(* Logix 5000 project; controller BTS01 vendor 1 type 14 code 217 rev 32.14; software revision 32.04; part 3 of 15 *)
(* tags used below, declared in another part *)
   AG1101 : DTE_VFD;   // Tank 1100 Agitator
   AG1201 : DTE_VFD;   // Tank 1200 Agitator
   Alarm_Active : DINT;
   Alarm_TMR : TIMER[17,32];
   ALM_ENABLE : DINT[25];
   C02S01 : REAL[8];   // 5069-IF8
   C02S03 : INT;   // 5069-IB16
   C02S06 : INT;   // 5069-IB16
   CIP_1_ACTIVE_CIRCUIT : DINT;
   CIP_1_Circuit1_Prox_Mismatch : BOOL;
   CIP_1_Circuit1_Tank_Not_Empty : BOOL;
   CIP_1_Circuit2_Prox_Mismatch : BOOL;
   CIP_1_Circuit2_Tank_Not_Empty : BOOL;
   CIP_1_Circuit3_Prox_Mismatch : BOOL;
   CIP_1_Circuit4_Prox_Mismatch : BOOL;
   CIP_1_SEQ_CTU : COUNTER;   // CIP 1 SEQUENCE STEP COUNTER THIS IS THE SEQUENCE STEP CONTROL
   CIP_1_START_PB_HMI : BOOL;
   CIP_Cart_Comm_Failed : BOOL;
   HMI_Global_Alarm_Ack_PB : BOOL;
   HMIAlarms : DINT[25];   // Alarm Trigger Array
   HMIAlarmsMsg : STRING64[17,32];   // Alarm Descriptions to Match Alarm Trigger Array
   P1001 : DTE_VFD;   // Dressing Tank Fill Pump
   P1002 : DTE_VFD;   // Product Filler Fill Pump
   P1003 : DTE_VFD;   // CIP Return Pump
   P1004 : DTE_VFD;   // Filler CIP Return Pump

   V1007_CIP_ENABLE : BOOL;
   V1007_CIP_PULSE : BOOL;
   V1007_Desc : STRING;
   V1007_PIDName : STRING;
   V1101 : DTE_Air_Valve_v2 := (CMD := 1, OUT := 1, ALM_PRE := 7000, P := 1, M := 2, Allowed := 1, Status := 1, ITEMTAG := 1101, MOA_Mode := 1);   // Tank 1100 Fill Valve
   V1101_CIP_ENABLE : BOOL;
   V1101_CIP_PULSE : BOOL;
   V1101_Desc : STRING;
   V1101_PIDName : STRING;
   V1102 : DTE_Air_Valve_v2 := (ALM_PRE := 7000, M := 2, Allowed := 1, ITEMTAG := 1102, MOA_Mode := 1);   // Tank 1100 Discharge Valve
   V1102_CIP_ENABLE : BOOL;
   V1102_CIP_PULSE : BOOL;
   V1102_Desc : STRING;
   V1102_PIDName : STRING;
   V1103 : DTE_Air_Valve_v2 := (ALM_PRE := 7000, M := 2, Allowed := 1, ITEMTAG := 1103, MOA_Mode := 1);   // Tank 1100 Line Valve
   V1103_CIP_ENABLE : BOOL;
   V1103_CIP_PULSE : BOOL;
   V1103_Desc : STRING;
   V1103_PIDName : STRING;
   V1201 : DTE_Air_Valve_v2 := (TOFF_OUT_ACC := 1, ALM_PRE := 7000, M := 2, Allowed := 1, ITEMTAG := 1201, MOA_Mode := 1);   // Tank 1200 Fill Valve
   V1201_CIP_ENABLE : BOOL;
   V1201_CIP_PULSE : BOOL;
   V1201_Desc : STRING;
   V1201_PIDName : STRING;
   V1202 : DTE_Air_Valve_v2 := (ALM_PRE := 7000, M := 2, Allowed := 1, ITEMTAG := 1202, MOA_Mode := 1);   // Tank 1200 Discharge Valve
   V1202_CIP_ENABLE : BOOL;
   V1202_CIP_PULSE : BOOL;
   V1202_Desc : STRING;
   V1202_PIDName : STRING;
   V1203 : DTE_Air_Valve_v2 := (ALM_PRE := 7000, M := 2, Allowed := 1, ITEMTAG := 1203, MOA_Mode := 1);   // Tank 1200 Line Valve
   V1203_CIP_ENABLE : BOOL;
   V1203_CIP_PULSE : BOOL;
   V1203_Desc : STRING;
   V1203_PIDName : STRING;
   VFD1001_SCP : DTE_SCP_W_LIM := (Input_Max := 100.0, Scaled_Max := 100.0, Limit_En := 1);   // Bowl Chopper Disc Speed Reference
   VFD1002_SCP : DTE_SCP_W_LIM := (Input_Max := 100.0, Scaled_Max := 100.0, Limit_En := 1);   // Dressing Tank Disc Speed Reference
   VFD1003_SCP : DTE_SCP_W_LIM := (Input_Max := 100.0, Scaled_Max := 100.0, Limit_En := 1);   // CIP Return Pump Speed Reference
   VFD1004_SCP : DTE_SCP_W_LIM := (Input_Max := 100.0, Scaled_Max := 100.0, Limit_En := 1);   // Filler CIP Return Pump Speed Reference
   VFD1101_SCP : DTE_SCP_W_LIM := (Input_Max := 100.0, Scaled_Max := 100.0, Limit_En := 1);   // Tank 1100 Agitator Speed Reference
   VFD1201_SCP : DTE_SCP_W_LIM := (Input_Max := 100.0, Scaled_Max := 100.0, Limit_En := 1);   // Tank 1200 Agitator Speed Reference
   ZS1000_1_Ind : DINT;
   ZS1000_2_Ind : DINT;
   ZS1000_3_Ind : DINT;
   ZS1000_4_Ind : DINT := 3;
   ZS1000_5_Ind : DINT;
   ZS1001_1_Ind : DINT;
   ZS1001_2_Ind : DINT;
   ZS1001_3_Ind : DINT;
   ZS1001_4_Ind : DINT;
   ZS1001_5_Ind : DINT := 3;
   ZS1101_Ind : DINT;
   ZS1201_Ind : DINT;
END_VAR

PROGRAM Alarm   (* main routine Alarm_Main *)

ROUTINE Alarm_00   (* ladder *)
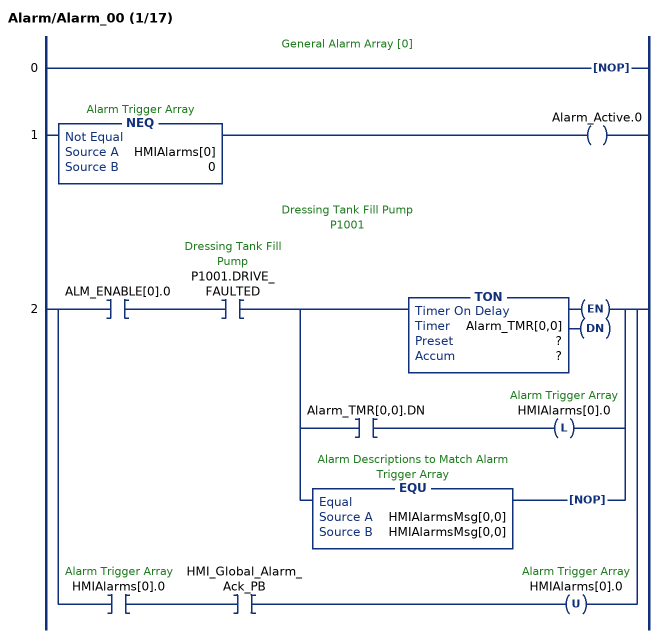
   // General Alarm Array [0]
   0: NOP();
   1: NEQ(HMIAlarms[0],0)OTE(Alarm_Active.0);
   // Dressing Tank Fill Pump
   // P1001
   2: [XIC(ALM_ENABLE[0].0) XIC(P1001.DRIVE_FAULTED) [TON(Alarm_TMR[0,0],?,?) ,XIC(Alarm_TMR[0,0].DN) OTL(HMIAlarms[0].0) ,EQU(HMIAlarmsMsg[0,0],HMIAlarmsMsg[0,0]) NOP() ] ,XIC(HMIAlarms[0].0) XIC(HMI_Global_Alarm_Ack_PB) OTU(HMIAlarms[0].0) ];
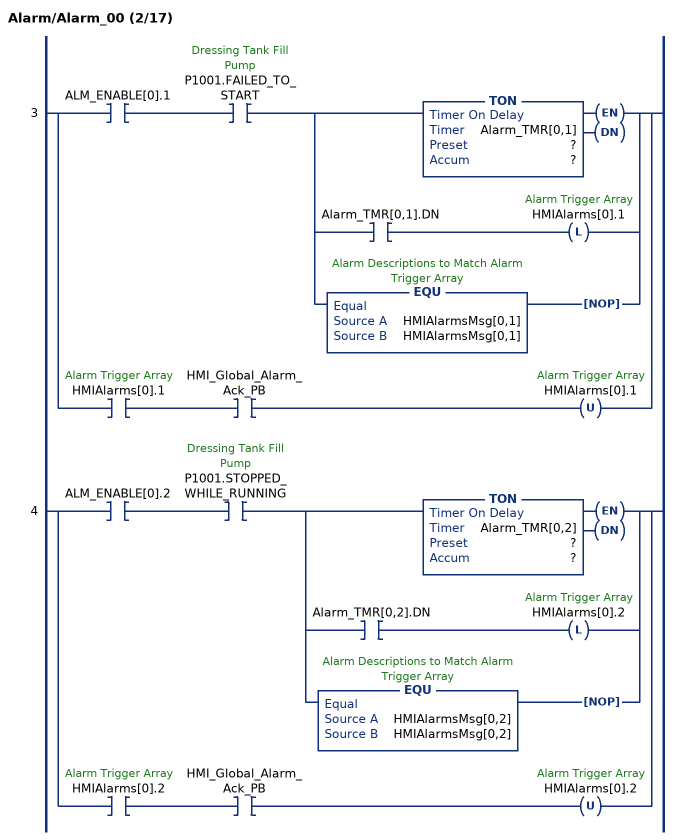
   3: [XIC(ALM_ENABLE[0].1) XIC(P1001.FAILED_TO_START) [TON(Alarm_TMR[0,1],?,?) ,XIC(Alarm_TMR[0,1].DN) OTL(HMIAlarms[0].1) ,EQU(HMIAlarmsMsg[0,1],HMIAlarmsMsg[0,1]) NOP() ] ,XIC(HMIAlarms[0].1) XIC(HMI_Global_Alarm_Ack_PB) OTU(HMIAlarms[0].1) ];
   4: [XIC(ALM_ENABLE[0].2) XIC(P1001.STOPPED_WHILE_RUNNING) [TON(Alarm_TMR[0,2],?,?) ,XIC(Alarm_TMR[0,2].DN) OTL(HMIAlarms[0].2) ,EQU(HMIAlarmsMsg[0,2],HMIAlarmsMsg[0,2]) NOP() ] ,XIC(HMIAlarms[0].2) XIC(HMI_Global_Alarm_Ack_PB) OTU(HMIAlarms[0].2) ];
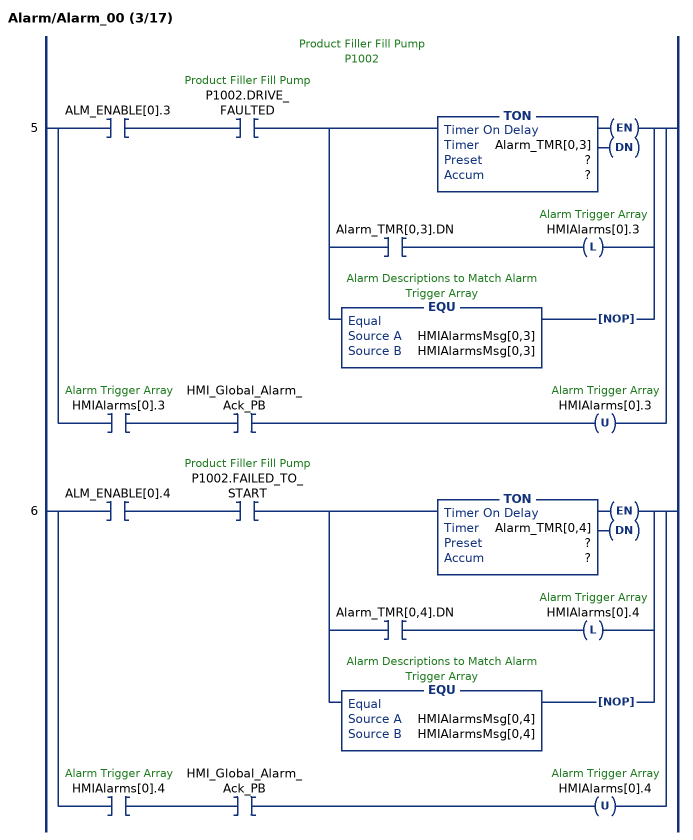
   // Product Filler Fill Pump
   // P1002
   5: [XIC(ALM_ENABLE[0].3) XIC(P1002.DRIVE_FAULTED) [TON(Alarm_TMR[0,3],?,?) ,XIC(Alarm_TMR[0,3].DN) OTL(HMIAlarms[0].3) ,EQU(HMIAlarmsMsg[0,3],HMIAlarmsMsg[0,3]) NOP() ] ,XIC(HMIAlarms[0].3) XIC(HMI_Global_Alarm_Ack_PB) OTU(HMIAlarms[0].3) ];
   6: [XIC(ALM_ENABLE[0].4) XIC(P1002.FAILED_TO_START) [TON(Alarm_TMR[0,4],?,?) ,XIC(Alarm_TMR[0,4].DN) OTL(HMIAlarms[0].4) ,EQU(HMIAlarmsMsg[0,4],HMIAlarmsMsg[0,4]) NOP() ] ,XIC(HMIAlarms[0].4) XIC(HMI_Global_Alarm_Ack_PB) OTU(HMIAlarms[0].4) ];
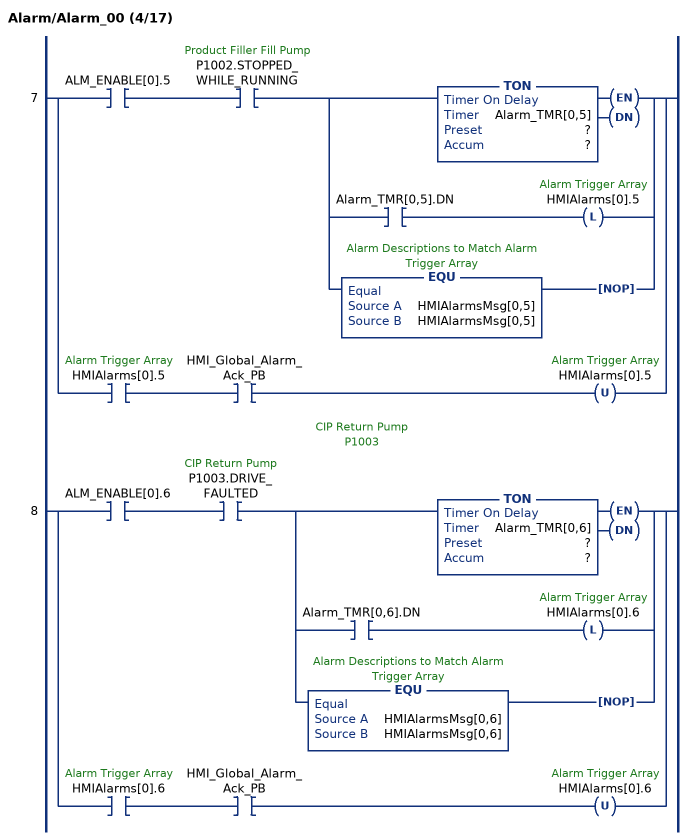
   7: [XIC(ALM_ENABLE[0].5) XIC(P1002.STOPPED_WHILE_RUNNING) [TON(Alarm_TMR[0,5],?,?) ,XIC(Alarm_TMR[0,5].DN) OTL(HMIAlarms[0].5) ,EQU(HMIAlarmsMsg[0,5],HMIAlarmsMsg[0,5]) NOP() ] ,XIC(HMIAlarms[0].5) XIC(HMI_Global_Alarm_Ack_PB) OTU(HMIAlarms[0].5) ];
   // CIP Return Pump
   // P1003
   8: [XIC(ALM_ENABLE[0].6) XIC(P1003.DRIVE_FAULTED) [TON(Alarm_TMR[0,6],?,?) ,XIC(Alarm_TMR[0,6].DN) OTL(HMIAlarms[0].6) ,EQU(HMIAlarmsMsg[0,6],HMIAlarmsMsg[0,6]) NOP() ] ,XIC(HMIAlarms[0].6) XIC(HMI_Global_Alarm_Ack_PB) OTU(HMIAlarms[0].6) ];
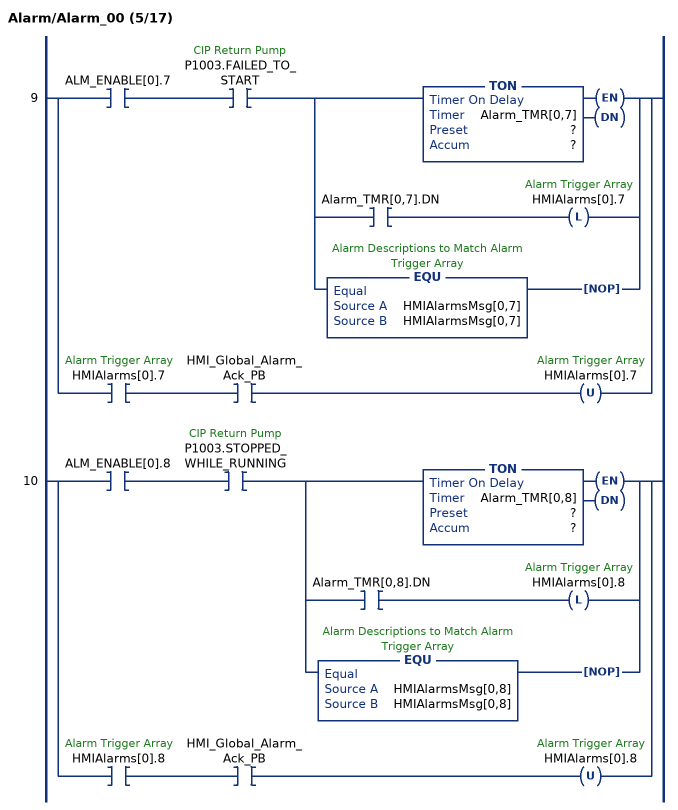
   9: [XIC(ALM_ENABLE[0].7) XIC(P1003.FAILED_TO_START) [TON(Alarm_TMR[0,7],?,?) ,XIC(Alarm_TMR[0,7].DN) OTL(HMIAlarms[0].7) ,EQU(HMIAlarmsMsg[0,7],HMIAlarmsMsg[0,7]) NOP() ] ,XIC(HMIAlarms[0].7) XIC(HMI_Global_Alarm_Ack_PB) OTU(HMIAlarms[0].7) ];
   10: [XIC(ALM_ENABLE[0].8) XIC(P1003.STOPPED_WHILE_RUNNING) [TON(Alarm_TMR[0,8],?,?) ,XIC(Alarm_TMR[0,8].DN) OTL(HMIAlarms[0].8) ,EQU(HMIAlarmsMsg[0,8],HMIAlarmsMsg[0,8]) NOP() ] ,XIC(HMIAlarms[0].8) XIC(HMI_Global_Alarm_Ack_PB) OTU(HMIAlarms[0].8) ];
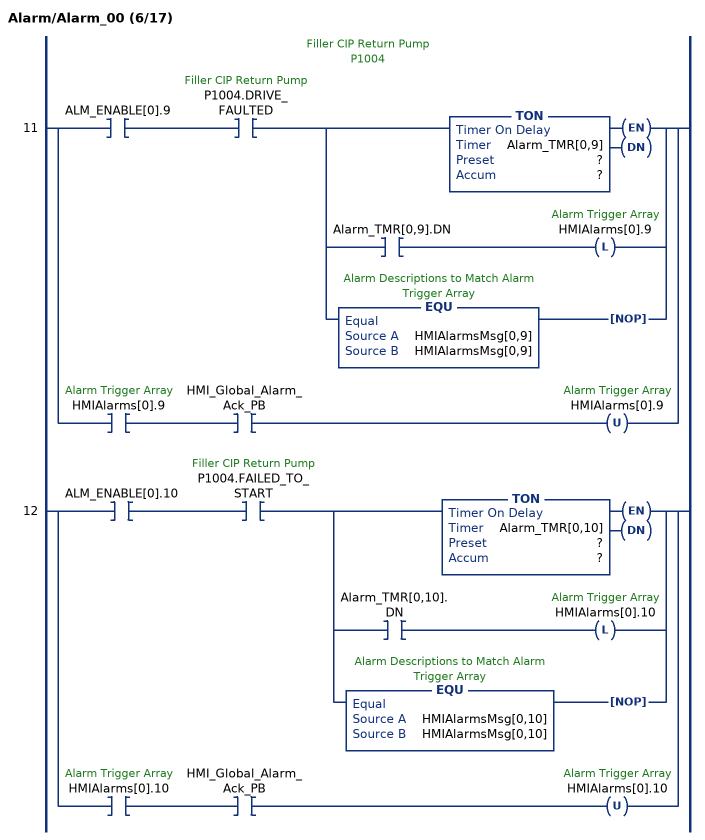
   // Filler CIP Return Pump
   // P1004
   11: [XIC(ALM_ENABLE[0].9) XIC(P1004.DRIVE_FAULTED) [TON(Alarm_TMR[0,9],?,?) ,XIC(Alarm_TMR[0,9].DN) OTL(HMIAlarms[0].9) ,EQU(HMIAlarmsMsg[0,9],HMIAlarmsMsg[0,9]) NOP() ] ,XIC(HMIAlarms[0].9) XIC(HMI_Global_Alarm_Ack_PB) OTU(HMIAlarms[0].9) ];
   12: [XIC(ALM_ENABLE[0].10) XIC(P1004.FAILED_TO_START) [TON(Alarm_TMR[0,10],?,?) ,XIC(Alarm_TMR[0,10].DN) OTL(HMIAlarms[0].10) ,EQU(HMIAlarmsMsg[0,10],HMIAlarmsMsg[0,10]) NOP() ] ,XIC(HMIAlarms[0].10) XIC(HMI_Global_Alarm_Ack_PB) OTU(HMIAlarms[0].10) ];
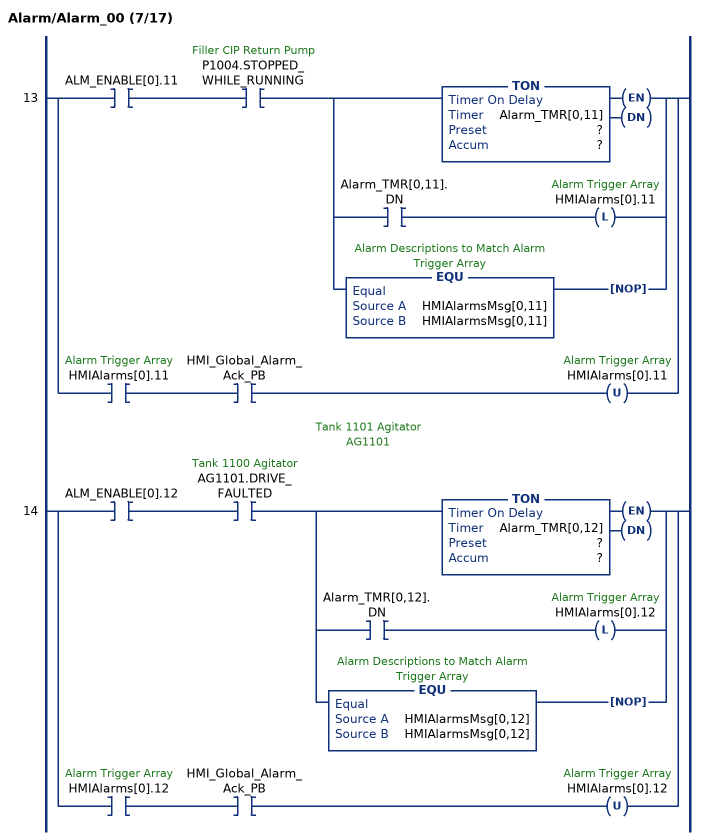
   13: [XIC(ALM_ENABLE[0].11) XIC(P1004.STOPPED_WHILE_RUNNING) [TON(Alarm_TMR[0,11],?,?) ,XIC(Alarm_TMR[0,11].DN) OTL(HMIAlarms[0].11) ,EQU(HMIAlarmsMsg[0,11],HMIAlarmsMsg[0,11]) NOP() ] ,XIC(HMIAlarms[0].11) XIC(HMI_Global_Alarm_Ack_PB) OTU(HMIAlarms[0].11) ];
   // Tank 1101 Agitator
   // AG1101
   14: [XIC(ALM_ENABLE[0].12) XIC(AG1101.DRIVE_FAULTED) [TON(Alarm_TMR[0,12],?,?) ,XIC(Alarm_TMR[0,12].DN) OTL(HMIAlarms[0].12) ,EQU(HMIAlarmsMsg[0,12],HMIAlarmsMsg[0,12]) NOP() ] ,XIC(HMIAlarms[0].12) XIC(HMI_Global_Alarm_Ack_PB) OTU(HMIAlarms[0].12) ];
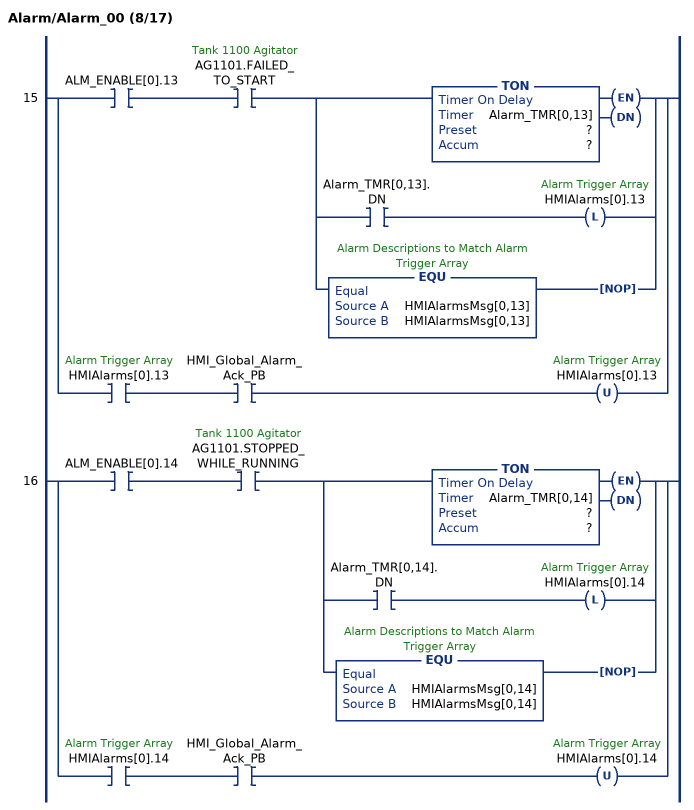
   15: [XIC(ALM_ENABLE[0].13) XIC(AG1101.FAILED_TO_START) [TON(Alarm_TMR[0,13],?,?) ,XIC(Alarm_TMR[0,13].DN) OTL(HMIAlarms[0].13) ,EQU(HMIAlarmsMsg[0,13],HMIAlarmsMsg[0,13]) NOP() ] ,XIC(HMIAlarms[0].13) XIC(HMI_Global_Alarm_Ack_PB) OTU(HMIAlarms[0].13) ];
   16: [XIC(ALM_ENABLE[0].14) XIC(AG1101.STOPPED_WHILE_RUNNING) [TON(Alarm_TMR[0,14],?,?) ,XIC(Alarm_TMR[0,14].DN) OTL(HMIAlarms[0].14) ,EQU(HMIAlarmsMsg[0,14],HMIAlarmsMsg[0,14]) NOP() ] ,XIC(HMIAlarms[0].14) XIC(HMI_Global_Alarm_Ack_PB) OTU(HMIAlarms[0].14) ];
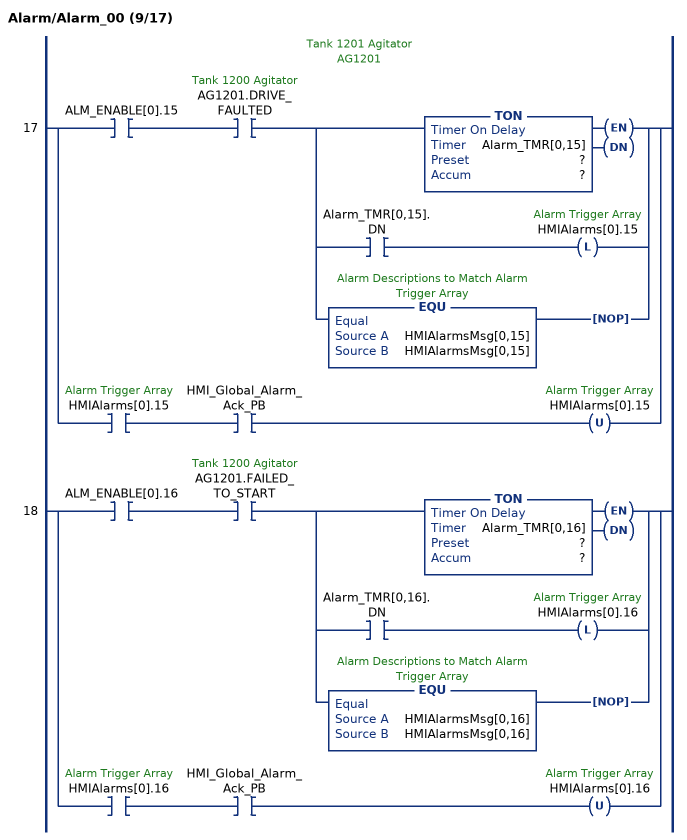
   // Tank 1201 Agitator
   // AG1201
   17: [XIC(ALM_ENABLE[0].15) XIC(AG1201.DRIVE_FAULTED) [TON(Alarm_TMR[0,15],?,?) ,XIC(Alarm_TMR[0,15].DN) OTL(HMIAlarms[0].15) ,EQU(HMIAlarmsMsg[0,15],HMIAlarmsMsg[0,15]) NOP() ] ,XIC(HMIAlarms[0].15) XIC(HMI_Global_Alarm_Ack_PB) OTU(HMIAlarms[0].15) ];
   18: [XIC(ALM_ENABLE[0].16) XIC(AG1201.FAILED_TO_START) [TON(Alarm_TMR[0,16],?,?) ,XIC(Alarm_TMR[0,16].DN) OTL(HMIAlarms[0].16) ,EQU(HMIAlarmsMsg[0,16],HMIAlarmsMsg[0,16]) NOP() ] ,XIC(HMIAlarms[0].16) XIC(HMI_Global_Alarm_Ack_PB) OTU(HMIAlarms[0].16) ];
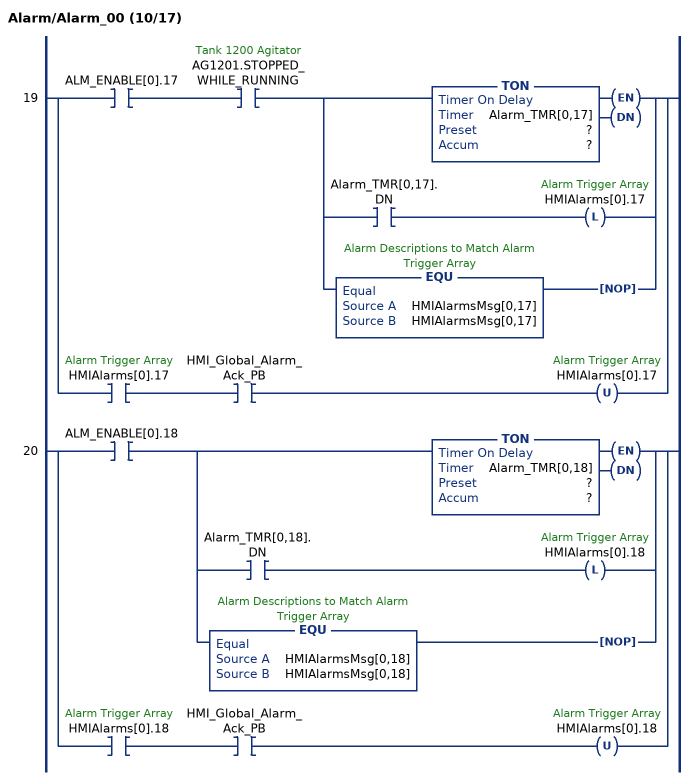
   19: [XIC(ALM_ENABLE[0].17) XIC(AG1201.STOPPED_WHILE_RUNNING) [TON(Alarm_TMR[0,17],?,?) ,XIC(Alarm_TMR[0,17].DN) OTL(HMIAlarms[0].17) ,EQU(HMIAlarmsMsg[0,17],HMIAlarmsMsg[0,17]) NOP() ] ,XIC(HMIAlarms[0].17) XIC(HMI_Global_Alarm_Ack_PB) OTU(HMIAlarms[0].17) ];
   20: [XIC(ALM_ENABLE[0].18) [TON(Alarm_TMR[0,18],?,?) ,XIC(Alarm_TMR[0,18].DN) OTL(HMIAlarms[0].18) ,EQU(HMIAlarmsMsg[0,18],HMIAlarmsMsg[0,18]) NOP() ] ,XIC(HMIAlarms[0].18) XIC(HMI_Global_Alarm_Ack_PB) OTU(HMIAlarms[0].18) ];
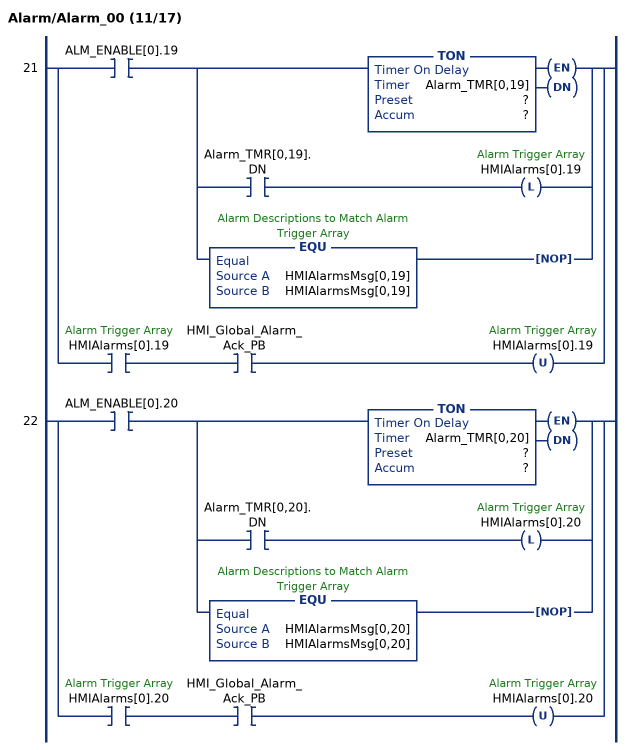
   21: [XIC(ALM_ENABLE[0].19) [TON(Alarm_TMR[0,19],?,?) ,XIC(Alarm_TMR[0,19].DN) OTL(HMIAlarms[0].19) ,EQU(HMIAlarmsMsg[0,19],HMIAlarmsMsg[0,19]) NOP() ] ,XIC(HMIAlarms[0].19) XIC(HMI_Global_Alarm_Ack_PB) OTU(HMIAlarms[0].19) ];
   22: [XIC(ALM_ENABLE[0].20) [TON(Alarm_TMR[0,20],?,?) ,XIC(Alarm_TMR[0,20].DN) OTL(HMIAlarms[0].20) ,EQU(HMIAlarmsMsg[0,20],HMIAlarmsMsg[0,20]) NOP() ] ,XIC(HMIAlarms[0].20) XIC(HMI_Global_Alarm_Ack_PB) OTU(HMIAlarms[0].20) ];
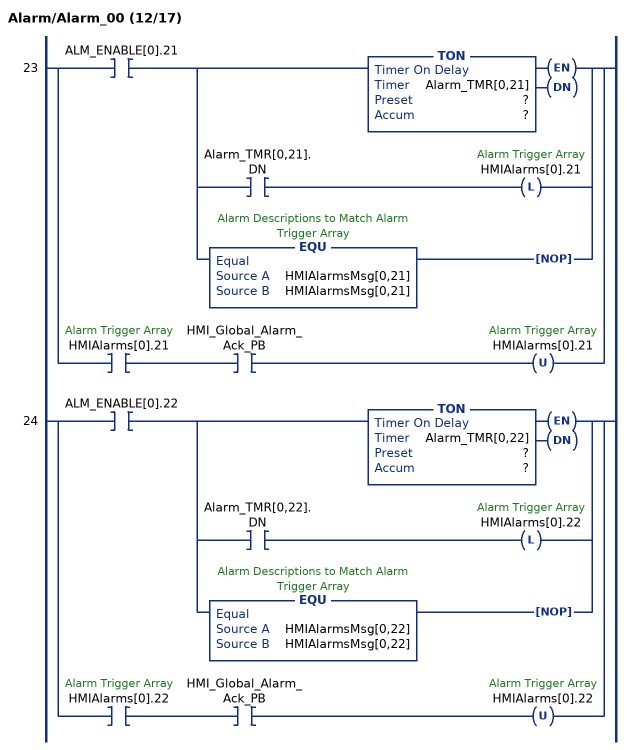
   23: [XIC(ALM_ENABLE[0].21) [TON(Alarm_TMR[0,21],?,?) ,XIC(Alarm_TMR[0,21].DN) OTL(HMIAlarms[0].21) ,EQU(HMIAlarmsMsg[0,21],HMIAlarmsMsg[0,21]) NOP() ] ,XIC(HMIAlarms[0].21) XIC(HMI_Global_Alarm_Ack_PB) OTU(HMIAlarms[0].21) ];
   24: [XIC(ALM_ENABLE[0].22) [TON(Alarm_TMR[0,22],?,?) ,XIC(Alarm_TMR[0,22].DN) OTL(HMIAlarms[0].22) ,EQU(HMIAlarmsMsg[0,22],HMIAlarmsMsg[0,22]) NOP() ] ,XIC(HMIAlarms[0].22) XIC(HMI_Global_Alarm_Ack_PB) OTU(HMIAlarms[0].22) ];
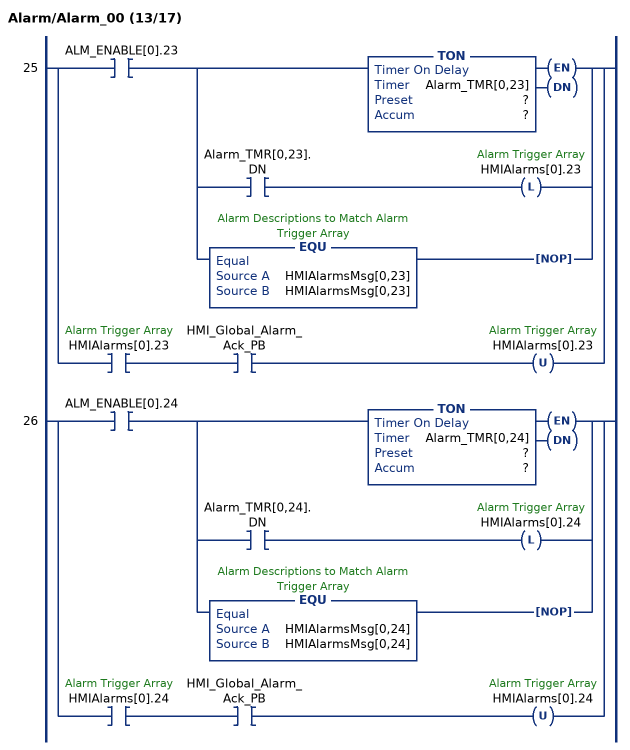
   25: [XIC(ALM_ENABLE[0].23) [TON(Alarm_TMR[0,23],?,?) ,XIC(Alarm_TMR[0,23].DN) OTL(HMIAlarms[0].23) ,EQU(HMIAlarmsMsg[0,23],HMIAlarmsMsg[0,23]) NOP() ] ,XIC(HMIAlarms[0].23) XIC(HMI_Global_Alarm_Ack_PB) OTU(HMIAlarms[0].23) ];
   26: [XIC(ALM_ENABLE[0].24) [TON(Alarm_TMR[0,24],?,?) ,XIC(Alarm_TMR[0,24].DN) OTL(HMIAlarms[0].24) ,EQU(HMIAlarmsMsg[0,24],HMIAlarmsMsg[0,24]) NOP() ] ,XIC(HMIAlarms[0].24) XIC(HMI_Global_Alarm_Ack_PB) OTU(HMIAlarms[0].24) ];
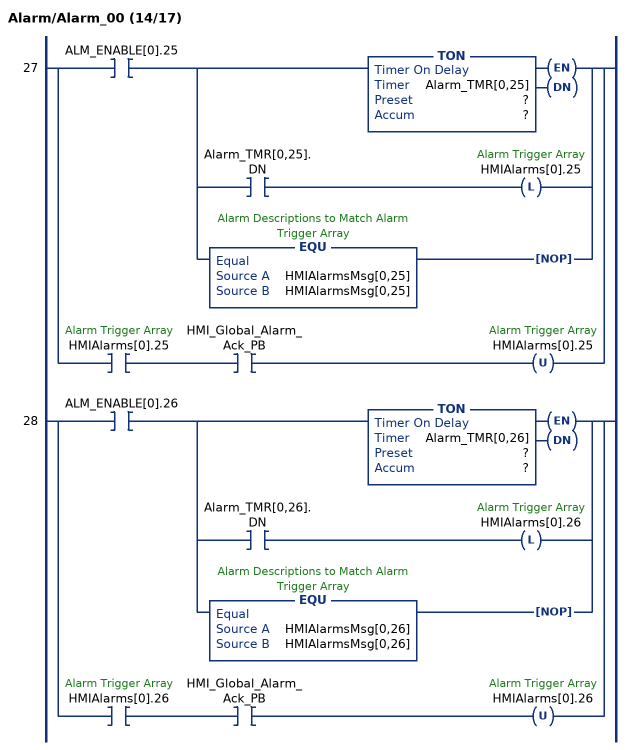
   27: [XIC(ALM_ENABLE[0].25) [TON(Alarm_TMR[0,25],?,?) ,XIC(Alarm_TMR[0,25].DN) OTL(HMIAlarms[0].25) ,EQU(HMIAlarmsMsg[0,25],HMIAlarmsMsg[0,25]) NOP() ] ,XIC(HMIAlarms[0].25) XIC(HMI_Global_Alarm_Ack_PB) OTU(HMIAlarms[0].25) ];
   28: [XIC(ALM_ENABLE[0].26) [TON(Alarm_TMR[0,26],?,?) ,XIC(Alarm_TMR[0,26].DN) OTL(HMIAlarms[0].26) ,EQU(HMIAlarmsMsg[0,26],HMIAlarmsMsg[0,26]) NOP() ] ,XIC(HMIAlarms[0].26) XIC(HMI_Global_Alarm_Ack_PB) OTU(HMIAlarms[0].26) ];
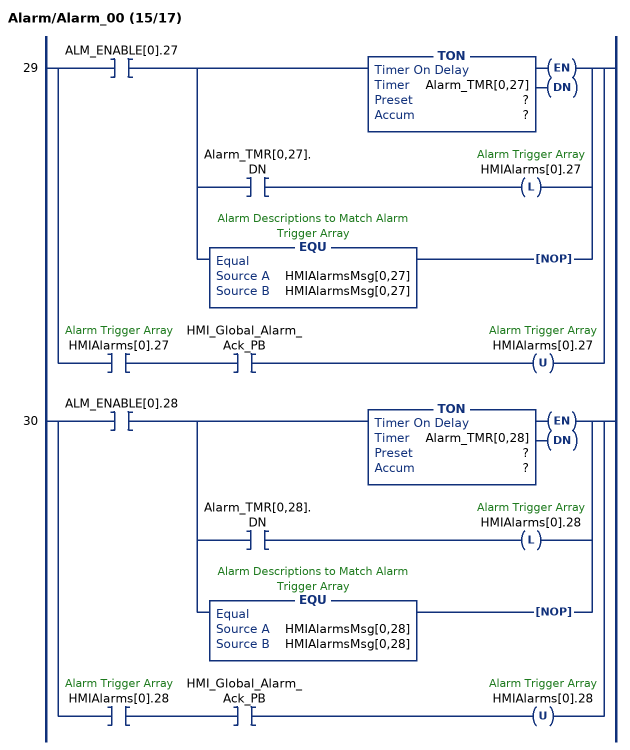
   29: [XIC(ALM_ENABLE[0].27) [TON(Alarm_TMR[0,27],?,?) ,XIC(Alarm_TMR[0,27].DN) OTL(HMIAlarms[0].27) ,EQU(HMIAlarmsMsg[0,27],HMIAlarmsMsg[0,27]) NOP() ] ,XIC(HMIAlarms[0].27) XIC(HMI_Global_Alarm_Ack_PB) OTU(HMIAlarms[0].27) ];
   30: [XIC(ALM_ENABLE[0].28) [TON(Alarm_TMR[0,28],?,?) ,XIC(Alarm_TMR[0,28].DN) OTL(HMIAlarms[0].28) ,EQU(HMIAlarmsMsg[0,28],HMIAlarmsMsg[0,28]) NOP() ] ,XIC(HMIAlarms[0].28) XIC(HMI_Global_Alarm_Ack_PB) OTU(HMIAlarms[0].28) ];
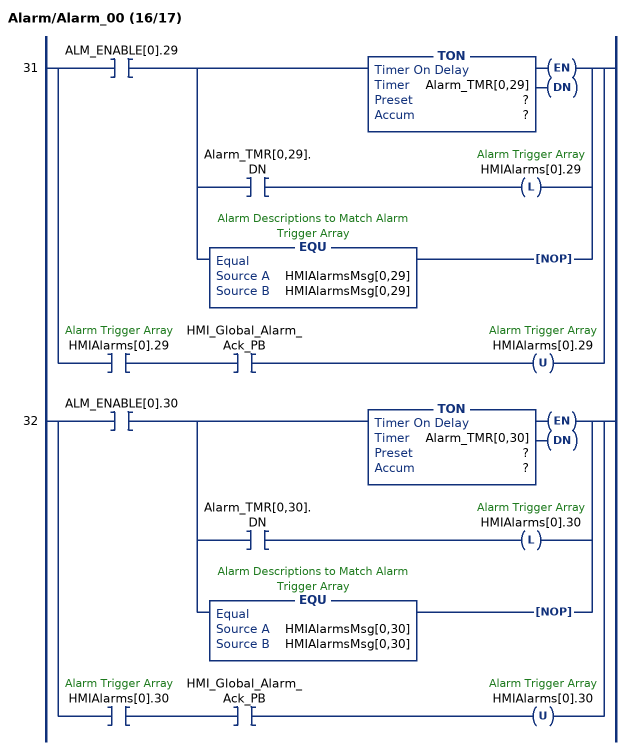
   31: [XIC(ALM_ENABLE[0].29) [TON(Alarm_TMR[0,29],?,?) ,XIC(Alarm_TMR[0,29].DN) OTL(HMIAlarms[0].29) ,EQU(HMIAlarmsMsg[0,29],HMIAlarmsMsg[0,29]) NOP() ] ,XIC(HMIAlarms[0].29) XIC(HMI_Global_Alarm_Ack_PB) OTU(HMIAlarms[0].29) ];
   32: [XIC(ALM_ENABLE[0].30) [TON(Alarm_TMR[0,30],?,?) ,XIC(Alarm_TMR[0,30].DN) OTL(HMIAlarms[0].30) ,EQU(HMIAlarmsMsg[0,30],HMIAlarmsMsg[0,30]) NOP() ] ,XIC(HMIAlarms[0].30) XIC(HMI_Global_Alarm_Ack_PB) OTU(HMIAlarms[0].30) ];
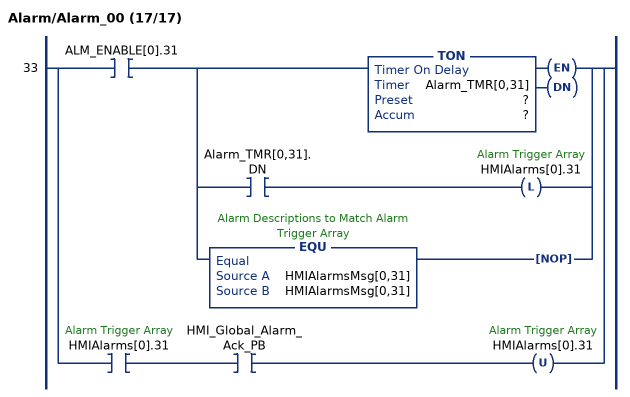
   33: [XIC(ALM_ENABLE[0].31) [TON(Alarm_TMR[0,31],?,?) ,XIC(Alarm_TMR[0,31].DN) OTL(HMIAlarms[0].31) ,EQU(HMIAlarmsMsg[0,31],HMIAlarmsMsg[0,31]) NOP() ] ,XIC(HMIAlarms[0].31) XIC(HMI_Global_Alarm_Ack_PB) OTU(HMIAlarms[0].31) ];
END_ROUTINE

ROUTINE Alarm_01   (* ladder *)
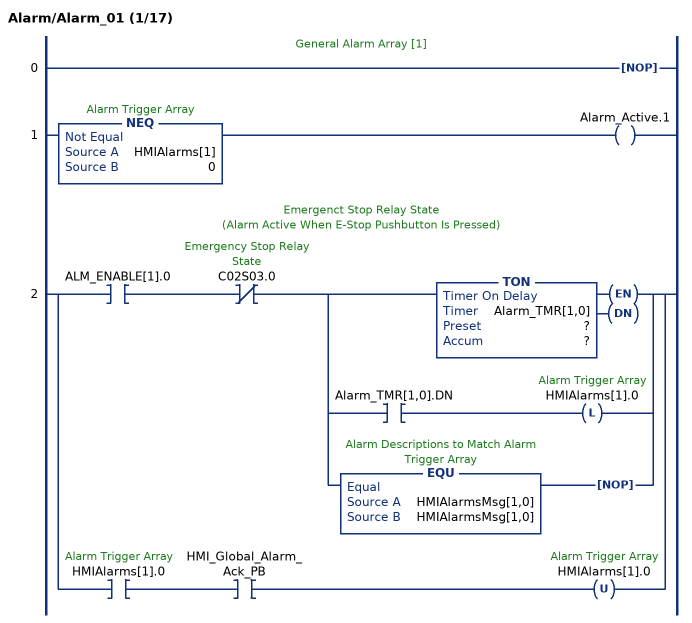
   // General Alarm Array [1]
   0: NOP();
   1: NEQ(HMIAlarms[1],0)OTE(Alarm_Active.1);
   // Emergenct Stop Relay State
   // (Alarm Active When E-Stop Pushbutton Is Pressed)
   2: [XIC(ALM_ENABLE[1].0) XIO(C02S03.0) [TON(Alarm_TMR[1,0],?,?) ,XIC(Alarm_TMR[1,0].DN) OTL(HMIAlarms[1].0) ,EQU(HMIAlarmsMsg[1,0],HMIAlarmsMsg[1,0]) NOP() ] ,XIC(HMIAlarms[1].0) XIC(HMI_Global_Alarm_Ack_PB) OTU(HMIAlarms[1].0) ];
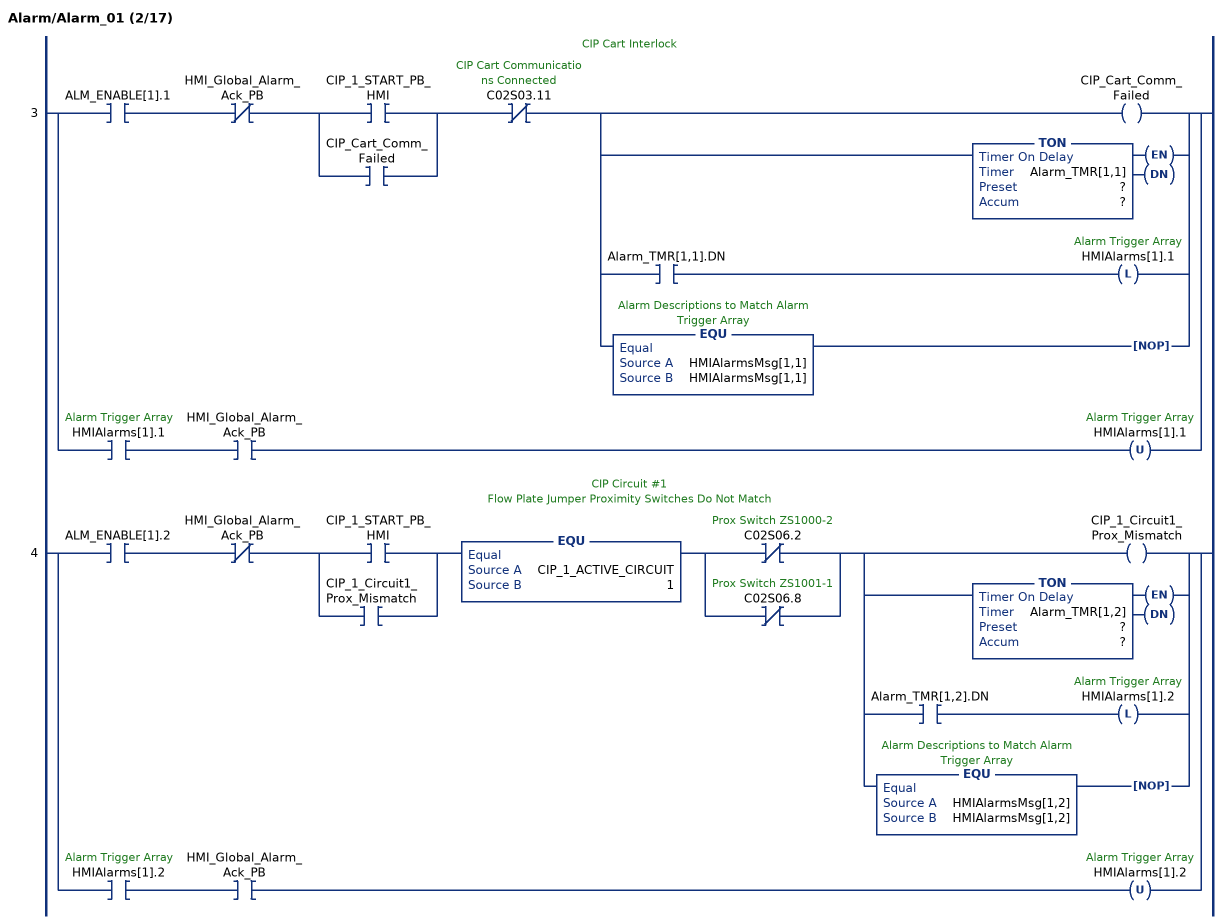
   // CIP Cart Interlock
   3: [XIC(ALM_ENABLE[1].1) XIO(HMI_Global_Alarm_Ack_PB) [XIC(CIP_1_START_PB_HMI) ,XIC(CIP_Cart_Comm_Failed) ] XIO(C02S03.11) [OTE(CIP_Cart_Comm_Failed) ,TON(Alarm_TMR[1,1],?,?) ,XIC(Alarm_TMR[1,1].DN) OTL(HMIAlarms[1].1) ,EQU(HMIAlarmsMsg[1,1],HMIAlarmsMsg[1,1]) NOP() ] ,XIC(HMIAlarms[1].1) XIC(HMI_Global_Alarm_Ack_PB) OTU(HMIAlarms[1].1) ];
   // CIP Circuit #1
   // Flow Plate Jumper Proximity Switches Do Not Match
   4: [XIC(ALM_ENABLE[1].2) XIO(HMI_Global_Alarm_Ack_PB) [XIC(CIP_1_START_PB_HMI) ,XIC(CIP_1_Circuit1_Prox_Mismatch) ] EQU(CIP_1_ACTIVE_CIRCUIT,1) [XIO(C02S06.2) ,XIO(C02S06.8) ] [OTE(CIP_1_Circuit1_Prox_Mismatch) ,TON(Alarm_TMR[1,2],?,?) ,XIC(Alarm_TMR[1,2].DN) OTL(HMIAlarms[1].2) ,EQU(HMIAlarmsMsg[1,2],HMIAlarmsMsg[1,2]) NOP() ] ,XIC(HMIAlarms[1].2) XIC(HMI_Global_Alarm_Ack_PB) OTU(HMIAlarms[1].2) ];
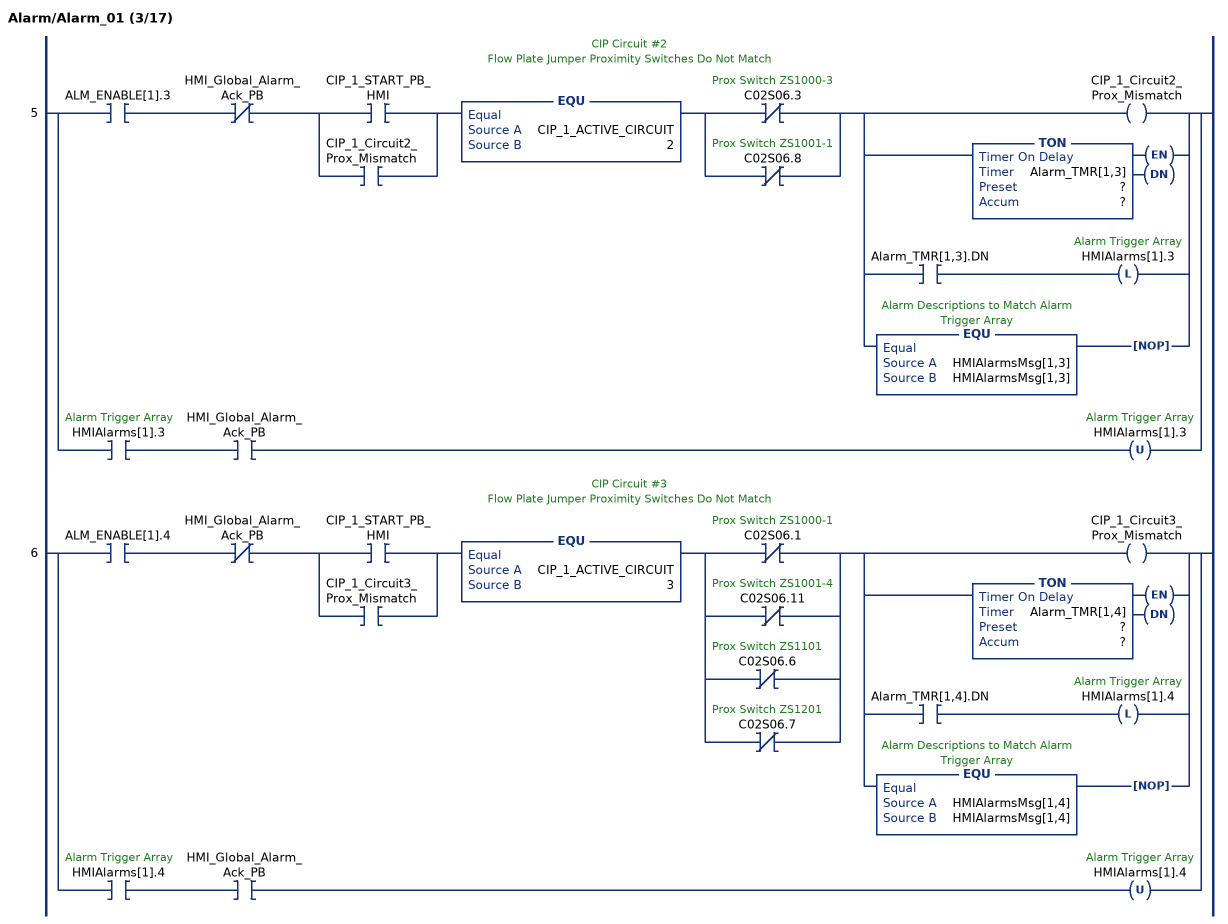
   // CIP Circuit #2
   // Flow Plate Jumper Proximity Switches Do Not Match
   5: [XIC(ALM_ENABLE[1].3) XIO(HMI_Global_Alarm_Ack_PB) [XIC(CIP_1_START_PB_HMI) ,XIC(CIP_1_Circuit2_Prox_Mismatch) ] EQU(CIP_1_ACTIVE_CIRCUIT,2) [XIO(C02S06.3) ,XIO(C02S06.8) ] [OTE(CIP_1_Circuit2_Prox_Mismatch) ,TON(Alarm_TMR[1,3],?,?) ,XIC(Alarm_TMR[1,3].DN) OTL(HMIAlarms[1].3) ,EQU(HMIAlarmsMsg[1,3],HMIAlarmsMsg[1,3]) NOP() ] ,XIC(HMIAlarms[1].3) XIC(HMI_Global_Alarm_Ack_PB) OTU(HMIAlarms[1].3) ];
   // CIP Circuit #3
   // Flow Plate Jumper Proximity Switches Do Not Match
   6: [XIC(ALM_ENABLE[1].4) XIO(HMI_Global_Alarm_Ack_PB) [XIC(CIP_1_START_PB_HMI) ,XIC(CIP_1_Circuit3_Prox_Mismatch) ] EQU(CIP_1_ACTIVE_CIRCUIT,3) [XIO(C02S06.1) ,XIO(C02S06.11) ,XIO(C02S06.6) ,XIO(C02S06.7) ] [OTE(CIP_1_Circuit3_Prox_Mismatch) ,TON(Alarm_TMR[1,4],?,?) ,XIC(Alarm_TMR[1,4].DN) OTL(HMIAlarms[1].4) ,EQU(HMIAlarmsMsg[1,4],HMIAlarmsMsg[1,4]) NOP() ] ,XIC(HMIAlarms[1].4) XIC(HMI_Global_Alarm_Ack_PB) OTU(HMIAlarms[1].4) ];
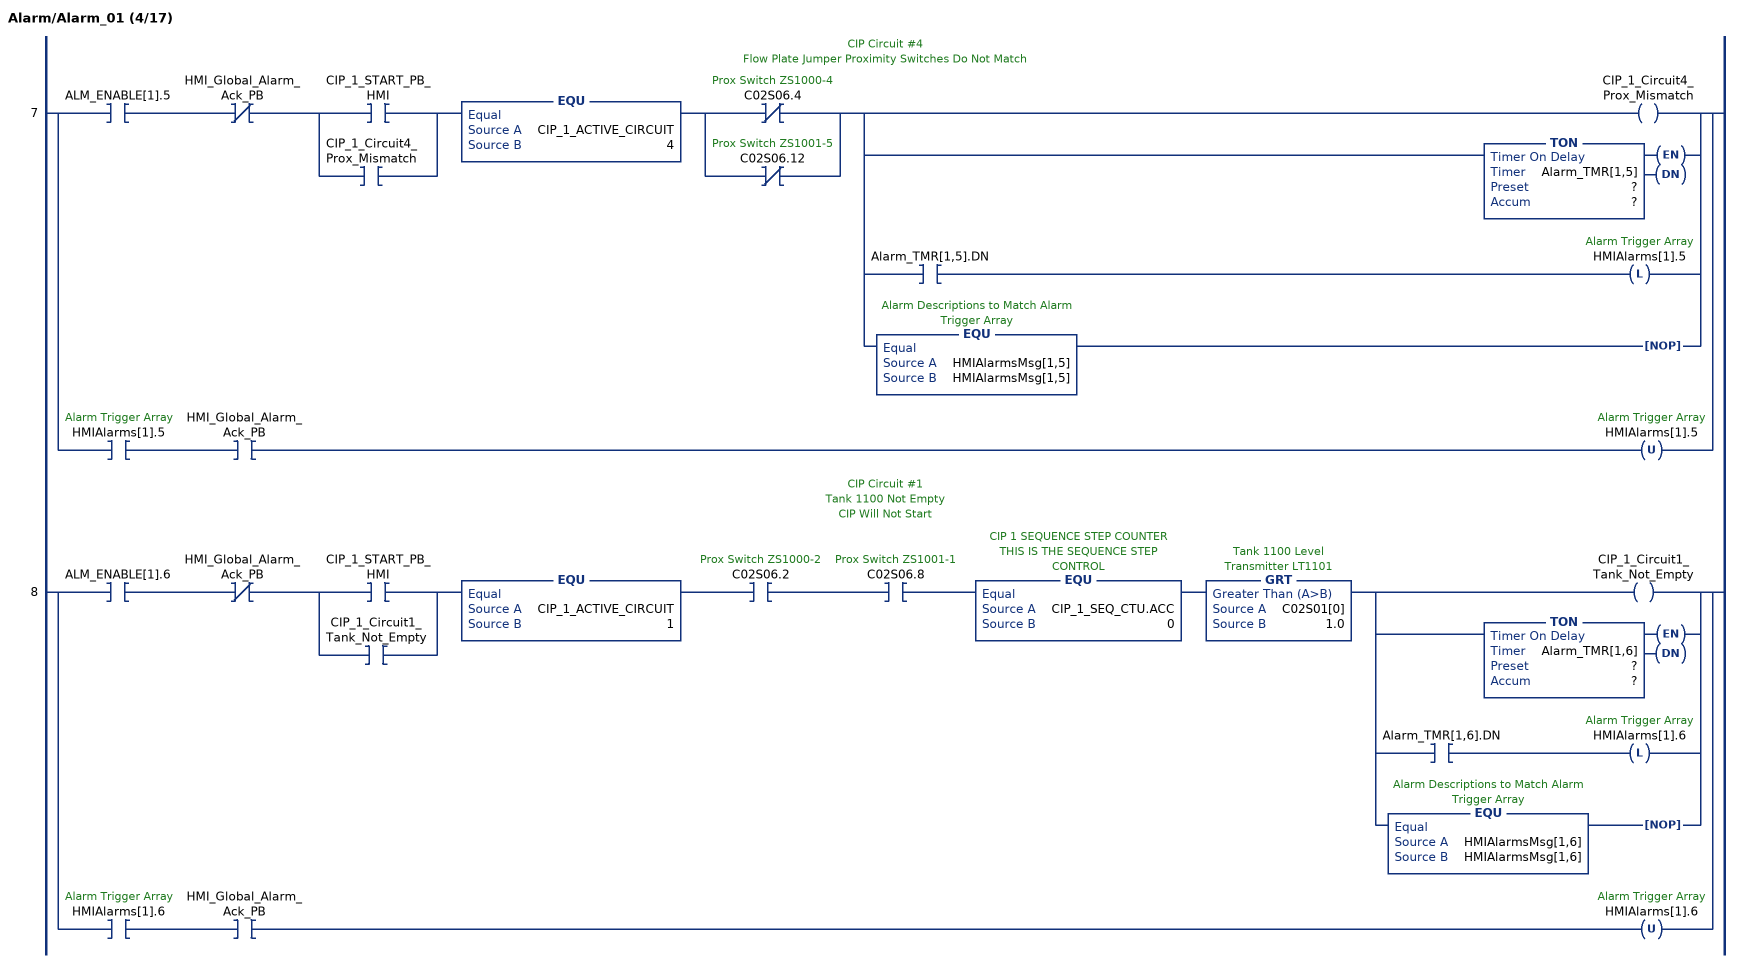
   // CIP Circuit #4
   // Flow Plate Jumper Proximity Switches Do Not Match
   7: [XIC(ALM_ENABLE[1].5) XIO(HMI_Global_Alarm_Ack_PB) [XIC(CIP_1_START_PB_HMI) ,XIC(CIP_1_Circuit4_Prox_Mismatch) ] EQU(CIP_1_ACTIVE_CIRCUIT,4) [XIO(C02S06.4) ,XIO(C02S06.12) ] [OTE(CIP_1_Circuit4_Prox_Mismatch) ,TON(Alarm_TMR[1,5],?,?) ,XIC(Alarm_TMR[1,5].DN) OTL(HMIAlarms[1].5) ,EQU(HMIAlarmsMsg[1,5],HMIAlarmsMsg[1,5]) NOP() ] ,XIC(HMIAlarms[1].5) XIC(HMI_Global_Alarm_Ack_PB) OTU(HMIAlarms[1].5) ];
   // CIP Circuit #1
   // Tank 1100 Not Empty
   // CIP Will Not Start
   8: [XIC(ALM_ENABLE[1].6) XIO(HMI_Global_Alarm_Ack_PB) [XIC(CIP_1_START_PB_HMI) ,XIC(CIP_1_Circuit1_Tank_Not_Empty) ] EQU(CIP_1_ACTIVE_CIRCUIT,1) XIC(C02S06.2) XIC(C02S06.8) EQU(CIP_1_SEQ_CTU.ACC,0) GRT(C02S01[0],1.0) [OTE(CIP_1_Circuit1_Tank_Not_Empty) ,TON(Alarm_TMR[1,6],?,?) ,XIC(Alarm_TMR[1,6].DN) OTL(HMIAlarms[1].6) ,EQU(HMIAlarmsMsg[1,6],HMIAlarmsMsg[1,6]) NOP() ] ,XIC(HMIAlarms[1].6) XIC(HMI_Global_Alarm_Ack_PB) OTU(HMIAlarms[1].6) ];
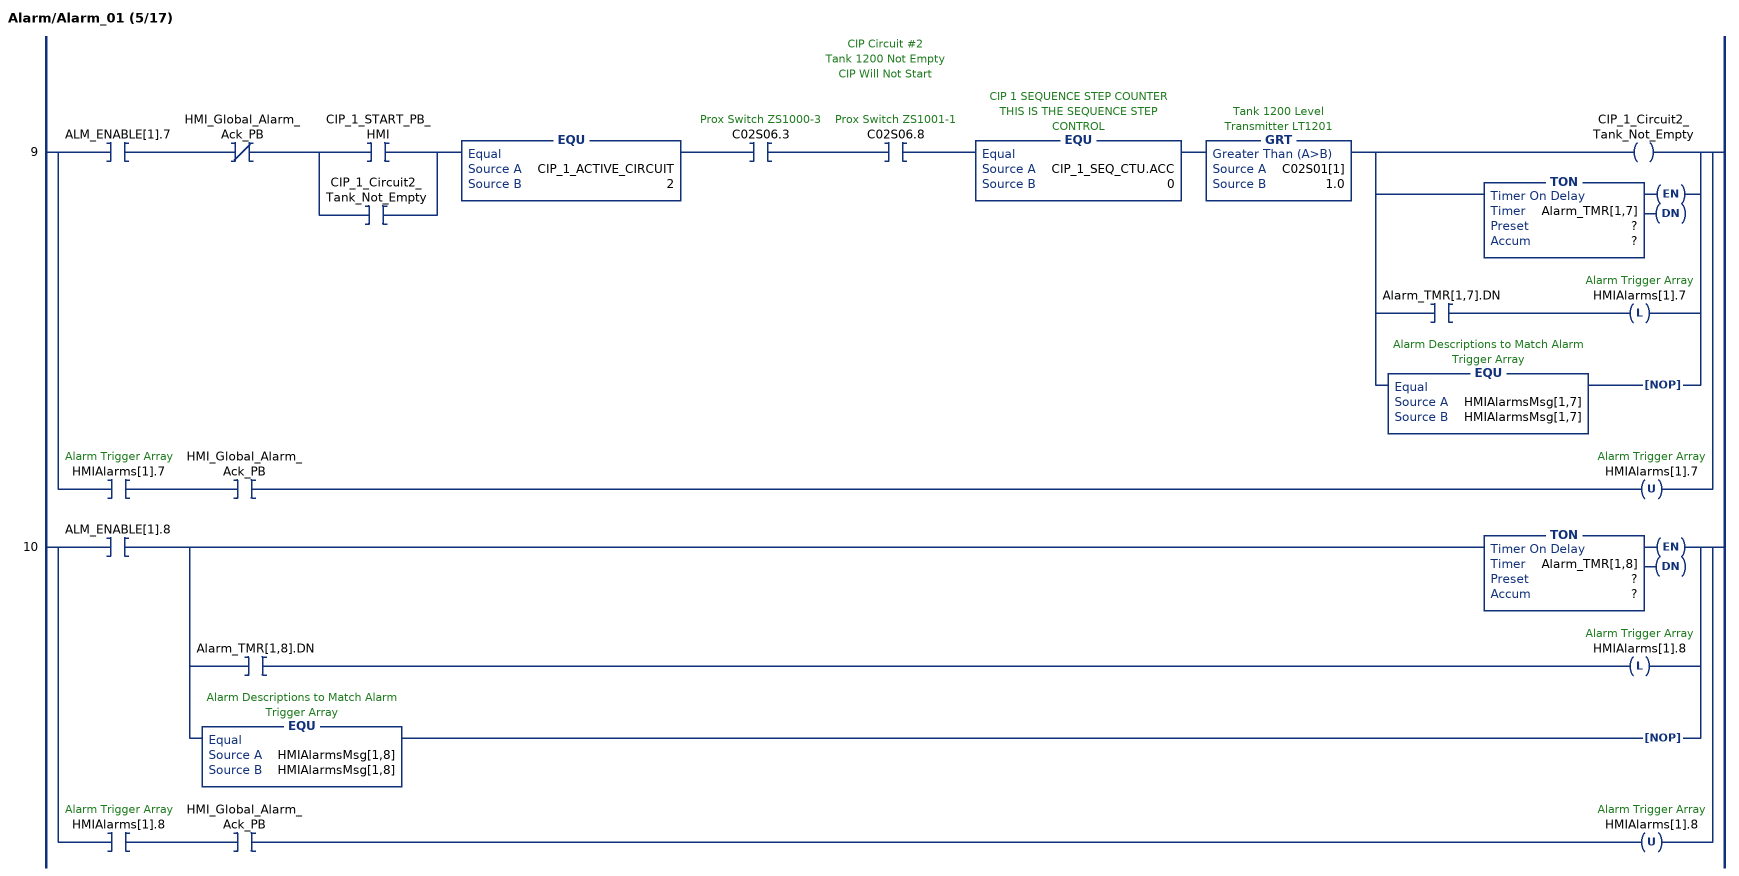
   // CIP Circuit #2
   // Tank 1200 Not Empty
   // CIP Will Not Start
   9: [XIC(ALM_ENABLE[1].7) XIO(HMI_Global_Alarm_Ack_PB) [XIC(CIP_1_START_PB_HMI) ,XIC(CIP_1_Circuit2_Tank_Not_Empty) ] EQU(CIP_1_ACTIVE_CIRCUIT,2) XIC(C02S06.3) XIC(C02S06.8) EQU(CIP_1_SEQ_CTU.ACC,0) GRT(C02S01[1],1.0) [OTE(CIP_1_Circuit2_Tank_Not_Empty) ,TON(Alarm_TMR[1,7],?,?) ,XIC(Alarm_TMR[1,7].DN) OTL(HMIAlarms[1].7) ,EQU(HMIAlarmsMsg[1,7],HMIAlarmsMsg[1,7]) NOP() ] ,XIC(HMIAlarms[1].7) XIC(HMI_Global_Alarm_Ack_PB) OTU(HMIAlarms[1].7) ];
   10: [XIC(ALM_ENABLE[1].8) [TON(Alarm_TMR[1,8],?,?) ,XIC(Alarm_TMR[1,8].DN) OTL(HMIAlarms[1].8) ,EQU(HMIAlarmsMsg[1,8],HMIAlarmsMsg[1,8]) NOP() ] ,XIC(HMIAlarms[1].8) XIC(HMI_Global_Alarm_Ack_PB) OTU(HMIAlarms[1].8) ];
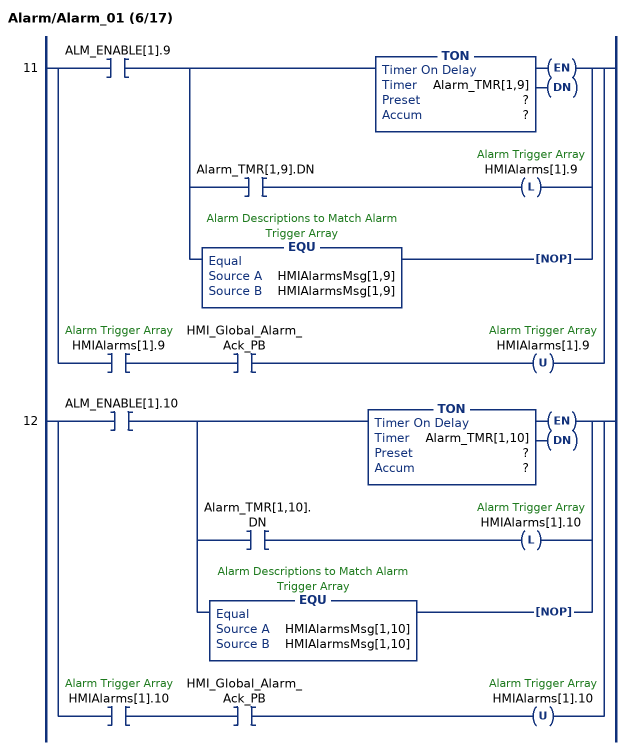
   11: [XIC(ALM_ENABLE[1].9) [TON(Alarm_TMR[1,9],?,?) ,XIC(Alarm_TMR[1,9].DN) OTL(HMIAlarms[1].9) ,EQU(HMIAlarmsMsg[1,9],HMIAlarmsMsg[1,9]) NOP() ] ,XIC(HMIAlarms[1].9) XIC(HMI_Global_Alarm_Ack_PB) OTU(HMIAlarms[1].9) ];
   12: [XIC(ALM_ENABLE[1].10) [TON(Alarm_TMR[1,10],?,?) ,XIC(Alarm_TMR[1,10].DN) OTL(HMIAlarms[1].10) ,EQU(HMIAlarmsMsg[1,10],HMIAlarmsMsg[1,10]) NOP() ] ,XIC(HMIAlarms[1].10) XIC(HMI_Global_Alarm_Ack_PB) OTU(HMIAlarms[1].10) ];
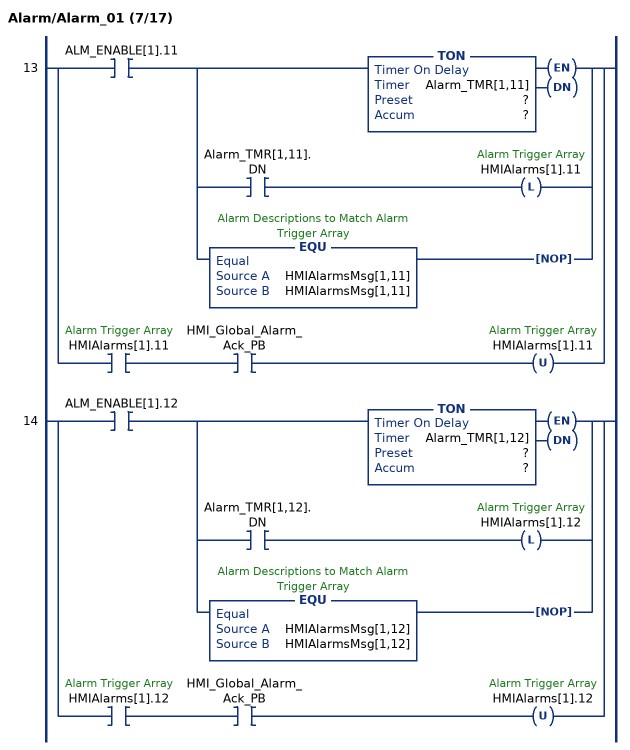
   13: [XIC(ALM_ENABLE[1].11) [TON(Alarm_TMR[1,11],?,?) ,XIC(Alarm_TMR[1,11].DN) OTL(HMIAlarms[1].11) ,EQU(HMIAlarmsMsg[1,11],HMIAlarmsMsg[1,11]) NOP() ] ,XIC(HMIAlarms[1].11) XIC(HMI_Global_Alarm_Ack_PB) OTU(HMIAlarms[1].11) ];
   14: [XIC(ALM_ENABLE[1].12) [TON(Alarm_TMR[1,12],?,?) ,XIC(Alarm_TMR[1,12].DN) OTL(HMIAlarms[1].12) ,EQU(HMIAlarmsMsg[1,12],HMIAlarmsMsg[1,12]) NOP() ] ,XIC(HMIAlarms[1].12) XIC(HMI_Global_Alarm_Ack_PB) OTU(HMIAlarms[1].12) ];
